// Mitsubishi GX Works2 project: 0624(슬라이드실린더_전진센서)   PLC: Q02/Q02H

PROGRAM MAIN
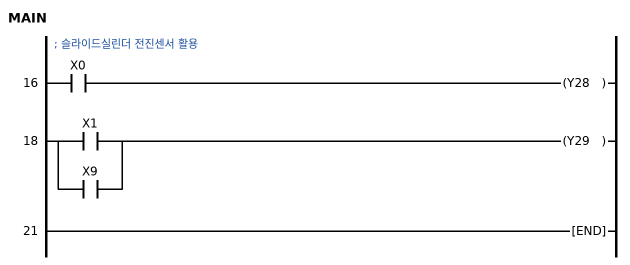
; 슬라이드실린더 전진센서 활용
16    LD      X0
      OUT     Y28
18    LD      X1
      OR      X9
      OUT     Y29
21    END
END_PROGRAM
